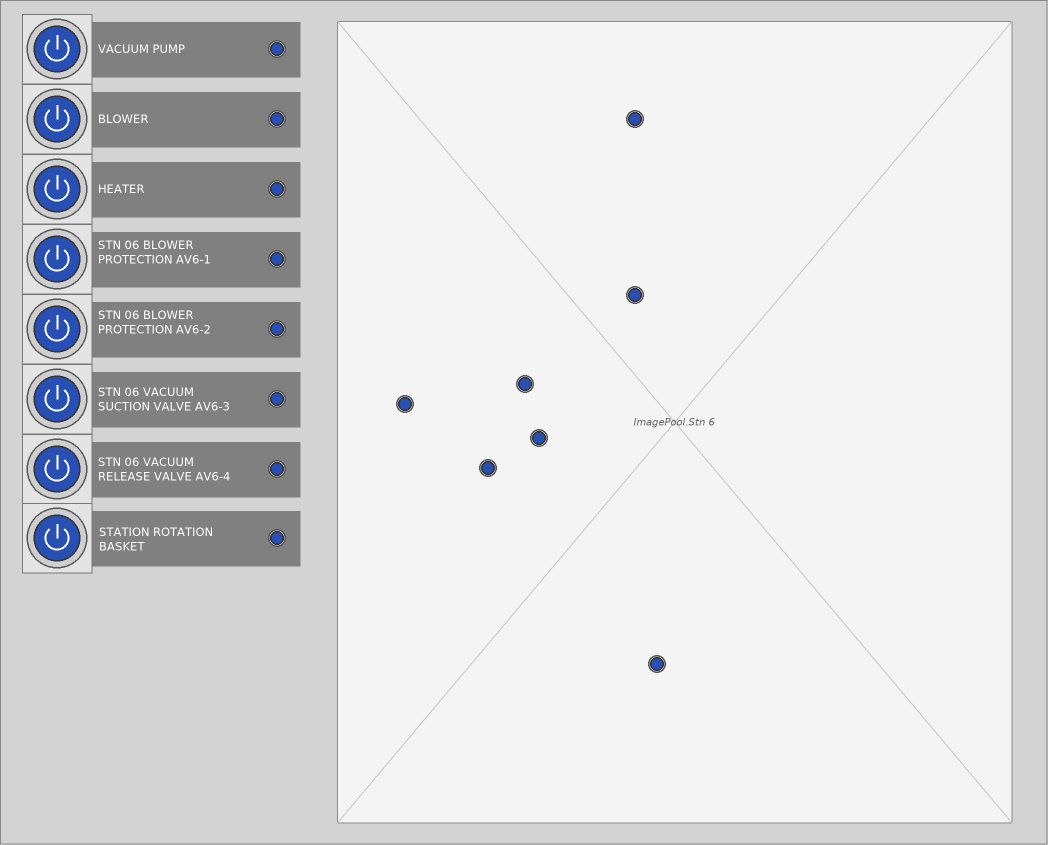
VISUALIZATION Recipe_Station06  // 1048x845
    Rectangle (0,0 1048x845)
    Image (337,21 675x802), image: ImagePool.Stn 6
    RoundedRectangle (61,22 239x55)
    Label (95,41 163x16), "VACUUM PUMP"
    Lamp1 (267,39 20x20), variable: DSScrMapSSUR.DsSubRecipeMemory.bOut11EnVacuumPump, style: Lamp-Lamp1-Blue
    PowerSwitch (22,14 70x70), variable: DSScrMapSSUR.DsSubRecipeMemory.bOut11EnVacuumPump, behaviour: TOGGLE, style: Switch-PowerSwitch-Blue
    RoundedRectangle (69,92 231x55)
    Label (95,111 151x16), "BLOWER"
    Lamp1 (267,109 20x20), variable: DSScrMapSSUR.DsSubRecipeMemory.bOut10EnBlower, style: Lamp-Lamp1-Blue
    PowerSwitch (22,84 70x70), variable: DSScrMapSSUR.DsSubRecipeMemory.bOut10EnBlower, behaviour: TOGGLE, style: Switch-PowerSwitch-Blue
    RoundedRectangle (61,162 239x55)
    Label (95,181 163x16), "HEATER"
    Lamp1 (267,179 20x20), variable: DSScrMapSSUR.DsSubRecipeMemory.bOut2EnProTankHeater, style: Lamp-Lamp1-Blue
    PowerSwitch (22,154 70x70), variable: DSScrMapSSUR.DsSubRecipeMemory.bOut2EnProTankHeater, behaviour: TOGGLE, style: Switch-PowerSwitch-Blue
    RoundedRectangle (69,232 231x55)
    Label (95,242 151x35), "STN 06 BLOWER PROTECTION AV6-1"
    Lamp1 (267,249 20x20), variable: DSScrMapSSUR.DsSubRecipeMemory.bOut1ActValve1, style: Lamp-Lamp1-Blue
    PowerSwitch (22,224 70x70), variable: DSScrMapSSUR.DsSubRecipeMemory.bOut1ActValve1, behaviour: TOGGLE, style: Switch-PowerSwitch-Blue
    RoundedRectangle (69,302 231x55)
    Label (95,312 151x35), "STN 06 BLOWER PROTECTION AV6-2"
    Lamp1 (267,319 20x20), variable: DSScrMapSSUR.DsSubRecipeMemory.bOut2ActValve2, style: Lamp-Lamp1-Blue
    PowerSwitch (22,294 70x70), variable: DSScrMapSSUR.DsSubRecipeMemory.bOut2ActValve2, behaviour: TOGGLE, style: Switch-PowerSwitch-Blue
    RoundedRectangle (69,372 231x55)
    Label (95,382 151x35), "STN 06 VACUUM SUCTION VALVE AV6-3"
    Lamp1 (267,389 20x20), variable: DSScrMapSSUR.DsSubRecipeMemory.bOut3ActValve3, style: Lamp-Lamp1-Blue
    PowerSwitch (22,364 70x70), variable: DSScrMapSSUR.DsSubRecipeMemory.bOut3ActValve3, behaviour: TOGGLE, style: Switch-PowerSwitch-Blue
    RoundedRectangle (69,442 231x55)
    Label (95,452 151x35), "STN 06 VACUUM RELEASE VALVE AV6-4"
    Lamp1 (267,459 20x20), variable: DSScrMapSSUR.DsSubRecipeMemory.bOut4ActValve4, style: Lamp-Lamp1-Blue
    PowerSwitch (22,434 70x70), variable: DSScrMapSSUR.DsSubRecipeMemory.bOut4ActValve4, behaviour: TOGGLE, style: Switch-PowerSwitch-Blue
    Lamp1 (647,654 20x20), variable: DSScrMapSSUR.DsSubRecipeMemory.bOut11EnVacuumPump, style: Lamp-Lamp1-Blue
    Lamp1 (529,428 20x20), variable: DSScrMapSSUR.DsSubRecipeMemory.bOut10EnBlower, style: Lamp-Lamp1-Blue
    Lamp1 (478,458 20x20), variable: DSScrMapSSUR.DsSubRecipeMemory.bOut2EnProTankHeater, style: Lamp-Lamp1-Blue
    Lamp1 (515,374 20x20), variable: DSScrMapSSUR.DsSubRecipeMemory.bOut2ActValve2, style: Lamp-Lamp1-Blue
    Lamp1 (625,285 20x20), variable: DSScrMapSSUR.DsSubRecipeMemory.bOut3ActValve3, style: Lamp-Lamp1-Blue
    Lamp1 (625,109 20x20), variable: DSScrMapSSUR.DsSubRecipeMemory.bOut4ActValve4, style: Lamp-Lamp1-Blue
    Lamp1 (395,394 20x20), variable: DSScrMapSSUR.DsSubRecipeMemory.bOut1ActValve1, style: Lamp-Lamp1-Blue
    RoundedRectangle (69,511 231x55)
    Label (96,525 151x29), "STATION ROTATION BASKET"
    Lamp1 (267,528 20x20), variable: DSScrMapSSUR.DsSubRecipeMemory.bOut14EnInstrument3, style: Lamp-Lamp1-Blue
    PowerSwitch (22,503 70x70), variable: DSScrMapSSUR.DsSubRecipeMemory.bOut14EnInstrument3, behaviour: TOGGLE, style: Switch-PowerSwitch-Blue
END_VISUALIZATION

(* stored: Version 1.1.0.1, ProductVersion 3.1.4024.12
   Visu Recipe_Station06: Id {edf221fa-e31a-43d9-9202-65bc78de9add} *)
